{attribute 'no_check'}
FUNCTION_BLOCK IOFcCom (* Frequence Converter IO Com *)
VAR_INPUT
	StartLeft												:	BOOL := FALSE;
	StartRight												:	BOOL := FALSE;
	InAck													:	BOOL := TRUE;
	Velo													:	LREAL := 0.0;
	VeloMin													:	LREAL := 0.0;
	VeloMax													:	LREAL := 100.0;
	FeedLeft												:	BOOL := TRUE;
	FeedRight												:	BOOL := TRUE;
	Contactor												:	BOOL;(* wenn vorhanden *)
	PT_DelBreak												:	TIME := T#1000MS;
	PT_DelEnable											:	TIME := T#1000MS;
	ProtSwitchOK											: 	FUSE;
	FuseBreakOK												: 	FUSE;
END_VAR         								
VAR_OUTPUT      								
	Ready											AT  %I* : 	BOOL := TRUE;
	Error											AT  %I* : 	BOOL := FALSE;
	Busy													:	BOOL;
{attribute 'displaymode':='binary'}
	Status													:	BYTE;
END_VAR
VAR (* IO Internal *)
	_SetValue										AT  %Q* : 	INT;
	_Reset											AT  %Q* :	BOOL;
	_Enable											AT  %Q* :	BOOL;
	_StartLeft										AT  %Q* :	BOOL;
	_StartRight										AT  %Q* :	BOOL;
	_Break											AT  %Q* :	BOOL; (* if available *)
	_Contactor										AT  %Q* :	BOOL;
END_VAR             								
VAR                 								
	TOF_Break												:	TOF;
	TOF_Enable												:	TOF;
	AckIntern												:	BOOL;
	BreakOpenIntern											:	BOOL;
END_VAR

(* Com FC IO 										 		V1.3	*)
(********************************************************************)

(* Protection Switch ************************************************)
	IF InAck 
	THEN 
		Ack(); 
	END_IF

	ProtSwitchOK(
		Force	:= ,
		Invert	:= ,
		InAck 	:= AckIntern,
		Q		=> ,
		Event 	=> ,
		INPUT 	=> );
		
	FuseBreakOK(InAck := AckIntern); (* same parameter like ProtSwitch *)

(* Contactor ********************************************************)
	_Contactor 												:= Contactor AND ProtSwitchOK.Q AND FuseBreakOK.Q;
	
(* Start ********************************************)
	IF 	StartRight 
		AND NOT StartLeft
	THEN
		SetStartRight();
	ELSIF StartLeft 
		AND NOT StartRight
	THEN
		SetStartLeft();
	ELSE
		 SetStop();
   END_IF

(* Enable ****************************************************)
	TOF_Enable(	IN := _SetValue <> 0,
					PT := PT_DelEnable);

	_Enable 												:= TOF_Enable.Q AND Ready AND _Break;

(* setvalue standardization *********************************)
	IF VeloMax > VeloMin THEN
		IF Velo >= VeloMax THEN
			_SetValue 										:= 32767;
		ELSIF Velo < VeloMin                				
		THEN                                				
			_SetValue 										:= 0;
		ELSE                                				
			_SetValue										:=LREAL_TO_INT ((32767.0 / (VeloMax - VeloMin)) * (Velo - VeloMin));
		END_IF                              				
	ELSE                                    				
		_SetValue 											:= 0;
	END_IF                                  				

(* setvalue **************************************)
	IF _StartLeft THEN
		_SetValue 											:= ABS(_SetValue) * -1;
	ELSIF _StartRight THEN              			
		_SetValue 											:= ABS(_SetValue);
	ELSE                                			
		_SetValue 											:= 0;
	END_IF                              	

(* HmiStatus **************************************************)
	Status.0 												:= _StartLeft AND Ready AND _Contactor;
	Status.1 												:= _StartRight AND Ready AND _Contactor;
	Status.2 												:= FALSE;
	Status.3 												:= _Break;
	Status.4 												:= FeedLeft ;
	Status.5 												:= FeedRight;
	Status.6 												:= Ready;
	Status.7 												:= Error;
	                                				
(* Status ***********************************************************)
	Busy 													:= TOF_Enable.Q AND TOF_Break.ET <= MAX(T#500MS,TOF_Break.PT) - T#500MS ;
	
(* Break ************************************************************)
	TOF_Break(	IN := _SetValue <> 0,
					PT := PT_DelBreak);

	IF _SetValue <> 0 
	THEN 
		BreakOpenIntern := FALSE; 
	END_IF

	_Break 													:= TOF_Break.Q AND Ready OR BreakOpenIntern;

(* Reset ***********************************************************)
	_Reset 													:= InAck OR AckIntern;
	AckIntern 												:= FALSE;

(**************************************************************)

METHOD PUBLIC Ack
VAR_INPUT
END_VAR
_Reset 														:= AckIntern 	:= TRUE;
END_METHOD

METHOD PUBLIC SetBreakClose
VAR_INPUT
END_VAR
BreakOpenIntern 											:= FALSE;
END_METHOD

METHOD PUBLIC SetBreakOpen
VAR_INPUT
END_VAR
BreakOpenIntern 							:= TRUE;
END_METHOD

METHOD PUBLIC SetContactorOFF
VAR_INPUT
END_VAR
Contactor 													:= FALSE;
SetStop();
END_METHOD

METHOD PUBLIC SetContactorON
VAR_INPUT
END_VAR
Contactor 													:= TRUE;
END_METHOD

METHOD PUBLIC SetStartLeft
VAR_INPUT
END_VAR
StartLeft 													:= TRUE; 
StartRight 													:= FALSE;
_StartLeft 													:= _Contactor AND Ready AND NOT Error AND FeedLeft;
END_METHOD

METHOD PUBLIC SetStartRight
VAR_INPUT
END_VAR
StartLeft 													:= FALSE; 
StartRight 													:= TRUE;
_StartRight 												:= _Contactor AND Ready AND NOT Error and FeedRight;
END_METHOD

METHOD PUBLIC SetStop
VAR_INPUT
END_VAR
StartLeft 													:= StartRight := _StartLeft := _StartRight := FALSE;
END_METHOD

END_FUNCTION_BLOCK

(* stored: Version 1.1.0.1, ProductVersion 3.1.4024.12
   POU IOFcCom: Id {2db019eb-408c-467e-8d26-0cce18b45cba}, SpecialFunc None
   Method Ack: Id {6a0f7972-dcdf-4de0-8c42-8191a4e4ccb9}
   Method SetBreakClose: Id {70780707-3221-4b65-91ef-bb50a6523e5e}
   Method SetBreakOpen: Id {0fe306ff-1961-4d37-9d83-afc912ebc7b4}
   Method SetContactorOFF: Id {a0b66d1d-adbe-454f-8752-c5656151d4b9}
   Method SetContactorON: Id {e082b2b1-8b41-4a63-aef8-a56e68289df3}
   Method SetStartLeft: Id {ae7e9107-9309-4d7b-8f91-b1bfcb1cc0a0}
   Method SetStartRight: Id {f84ae6ff-b7d2-4cc4-b150-69ad18ea2604}
   Method SetStop: Id {7c3e0c56-3f62-42db-b880-d750c2b08e2f} *)
